TYPE "VALVE_CMD"
VERSION : 0.1
   STRUCT
      Reset : Bool;   // Сброс отказов
      Open : Bool;   // Пуск
      Close : Bool;   // Стоп
      Auto : Bool;   // Авто режим (Дистанционный)
      Man : Bool;   // Ручной режим (Дистанционный)
      Cas : Bool;
   END_STRUCT;

END_TYPE

